// TIA Portal V17 export
// export: Created 2022-12-08T07:31:26.2167371Z, ExportSetting WithDefaults, DisplayName Totally Integrated Automation Portal, DisplayVersion V17 Update 5, DisplayName TIA Portal Openness, DisplayVersion V17 Update 5, DisplayName TIA Portal Version Control Interface, DisplayVersion V17, DisplayName Simotion SCOUT TIA, DisplayVersion 5.4.3.0, DisplayName SINAMICS Startdrive Advanced, DisplayVersion V17 SP1, DisplayName SINAMICS Startdrive G130, G150, S120, S150, SINAMICS MV, S210, DisplayVersion V17 SP1, DisplayName SINAMICS Startdrive G110M, G120, G120C, G120D, G120P, G115D, DisplayVersion V17 SP1, DisplayName STEP 7 Professional, DisplayVersion V17 Update 5, DisplayName STEP 7 Safety, DisplayVersion V17, DisplayName WinCC Advanced, DisplayVersion V17 Update 5
DATA_BLOCK "DB_BDE"   // DB700
AUTHOR : EconoPak GmbH
VERSION : 0.1
// stored: AutoNumber true, DBAccessibleFromOPCUA true, DBAccessibleFromWebserver true, InstanceOfName FB_BDE, InstanceOfType FB
"FB_BDE"
   // VAR_INPUT
   //    i_CountTotal_OK : DInt;
   //    i_CountTotal_NOK : DInt;
   //    i_CountTotal_In : DInt;
   // END_VAR
   // VAR_OUTPUT
   //    q_ProductionData : "UDT_BDE";
   // END_VAR
   // VAR_IN_OUT
   //    iq_InformationMessages : "UDT_Messages";
   //    iq_OperateMessages : "UDT_Messages";
   //    iq_FaultMessagesAbsolut : "UDT_Messages";
   //    iq_FaultMessagesCycleEnd : "UDT_Messages";
   //    iq_OMACGlobalData : "UDT_OMAC_GlobalData";
   // END_VAR
   // VAR
   //    stat_InformationMessages : "UDT_Messages";
   //    stat_OperateMessages : "UDT_Messages";
   //    stat_FaultMessagesAbsolut : "UDT_Messages";
   //    stat_FaultMessagesCycleEnd : "UDT_Messages";
   // END_VAR
BEGIN
END_DATA_BLOCK
